{attribute 'qualified_only'}
TYPE MotionlinxAI_Motor_Status :
(
	MOTOR_NOT_RUNNING_BRAKED := 0 ,
	MOTOR_NOT_RUNNING_UNBRAKED,
	MOTOR_RUNNING_CCW,
	MOTOR_RUNNING_CW
);
END_TYPE

(* stored: Version 1.1.0.1, ProductVersion 3.1.4024.16
   DUT MotionlinxAI_Motor_Status: Id {07721bff-f139-4c81-9fb2-daf6172eeabd} *)
